TYPE "MEStoPLC_PrintExchange_ext"
VERSION : 0.1
   STRUCT
      Load_PrintReqOK : Bool;
      Load_PrintReqNG : Bool;
      Load_PrintReqDone : Bool;
      Load_DataMatrixCheckOK : Bool;
      Load_DataMatrixCheckNG : Bool;
      Load_DataMatrixCheckDone : Bool;
      Spare : Bool;
      Spare_1 : Bool;
      SpareByte : Byte;
      SpareByte_1 : Byte;
   END_STRUCT;

END_TYPE

